FUNCTION F_LTrimEx : T_MaxString // removes n characters from start of string
VAR_INPUT
   n : UINT; 
   str : T_MaxString;
END_VAR
VAR
    Length : UINT;
END_VAR

Length := INT_TO_UINT(LEN(str));
IF n = 0 THEN
    F_LTrimEx := str;
ELSIF n < Length THEN
    MEMCPY(destAddr := ADR(F_LTrimEx),
           srcAddr  := ADR(str) + n,
           n        := Length - n + 1); // include null terminator
END_IF

END_FUNCTION

(* stored: Version 1.1.0.1, ProductVersion 3.1.4024.3
   POU F_LTrimEx: Id {b231ba14-158f-4b86-a454-3236e2e0f35d}, SpecialFunc None *)
